// Single-character string alias.
TYPE Ch : STRING(1); END_TYPE

(* stored: Version 1.1.0.1
   DUT Ch: Id {ddd91310-5dcc-459c-a150-49ad8e7e22bc} *)
